TYPE ST_LrealDataPoint :
STRUCT
	Timestamp	: ULINT;
	Value		: LREAL;
END_STRUCT
END_TYPE

(* stored: Version 1.1.0.1
   DUT ST_LrealDataPoint: Id {a6326554-b881-4532-9341-0b67289f57e2} *)
